// Mitsubishi GX Works2 project: Ex5   PLC: Q03UDV

PROGRAM MAIN
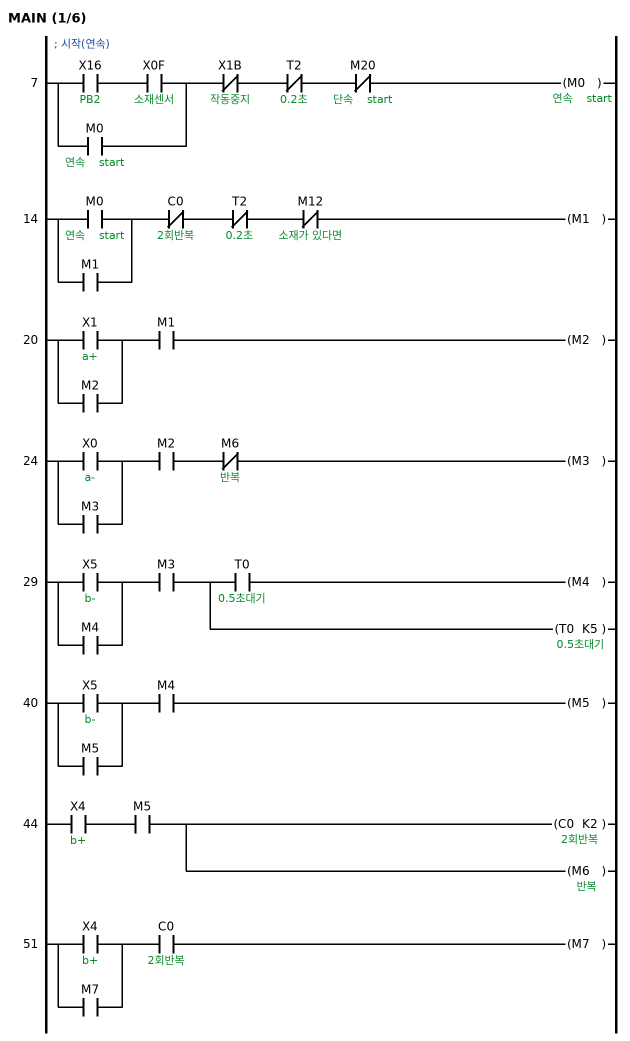
; 시작(연속)
7     LD      X16  ; PB2
      AND     X0F  ; 소재센서
      OR      M0  ; 연속    start
      ANI     X1B  ; 작동중지
      ANI     T2  ; 0.2초
      ANI     M20  ; 단속    start
      OUT     M0  ; 연속    start
14    LD      M0  ; 연속    start
      OR      M1
      ANI     C0  ; 2회반복
      ANI     T2  ; 0.2초
      ANI     M12  ; 소재가 있다면
      OUT     M1
20    LD      X1  ; a+
      OR      M2
      AND     M1
      OUT     M2
24    LD      X0  ; a-
      OR      M3
      AND     M2
      ANI     M6  ; 반복
      OUT     M3
29    LD      X5  ; b-
      OR      M4
      AND     M3
      MPS
      AND     T0  ; 0.5초대기
      OUT     M4
      MPP
      OUT     T0 K5  ; 0.5초대기
40    LD      X5  ; b-
      OR      M5
      AND     M4
      OUT     M5
44    LD      X4  ; b+
      AND     M5
      OUT     C0 K2  ; 2회반복
      OUT     M6  ; 반복
51    LD      X4  ; b+
      OR      M7
      AND     C0  ; 2회반복
      OUT     M7
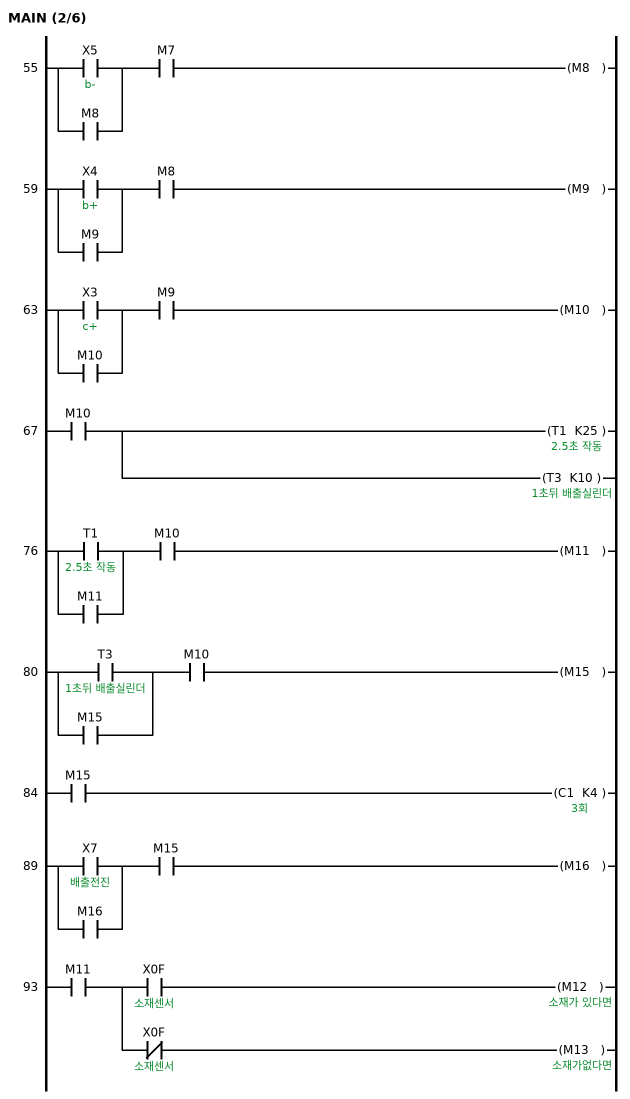
55    LD      X5  ; b-
      OR      M8
      AND     M7
      OUT     M8
59    LD      X4  ; b+
      OR      M9
      AND     M8
      OUT     M9
63    LD      X3  ; c+
      OR      M10
      AND     M9
      OUT     M10
67    LD      M10
      OUT     T1 K25  ; 2.5초 작동
      OUT     T3 K10  ; 1초뒤 배출실린더
76    LD      T1  ; 2.5초 작동
      OR      M11
      AND     M10
      OUT     M11
80    LD      T3  ; 1초뒤 배출실린더
      OR      M15
      AND     M10
      OUT     M15
84    LD      M15
      OUT     C1 K4  ; 3회
89    LD      X7  ; 배출전진
      OR      M16
      AND     M15
      OUT     M16
93    LD      M11
      MPS
      AND     X0F  ; 소재센서
      OUT     M12  ; 소재가 있다면
      MPP
      ANI     X0F  ; 소재센서
      OUT     M13  ; 소재가없다면
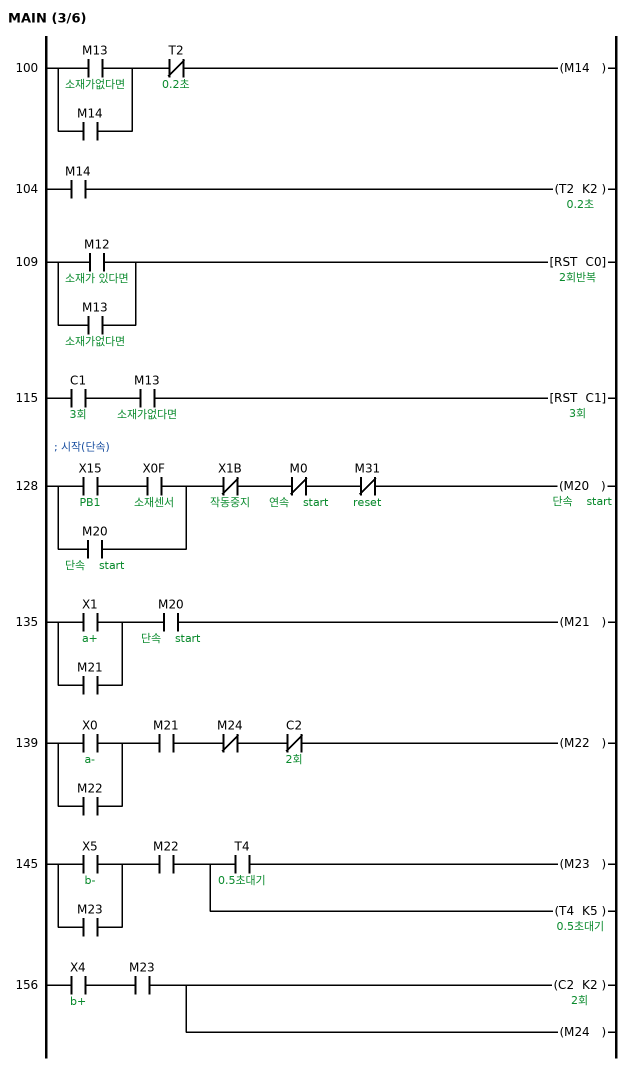
100   LD      M13  ; 소재가없다면
      OR      M14
      ANI     T2  ; 0.2초
      OUT     M14
104   LD      M14
      OUT     T2 K2  ; 0.2초
109   LD      M12  ; 소재가 있다면
      OR      M13  ; 소재가없다면
      RST     C0  ; 2회반복
115   LD      C1  ; 3회
      AND     M13  ; 소재가없다면
      RST     C1  ; 3회
; 시작(단속)
128   LD      X15  ; PB1
      AND     X0F  ; 소재센서
      OR      M20  ; 단속    start
      ANI     X1B  ; 작동중지
      ANI     M0  ; 연속    start
      ANI     M31  ; reset
      OUT     M20  ; 단속    start
135   LD      X1  ; a+
      OR      M21
      AND     M20  ; 단속    start
      OUT     M21
139   LD      X0  ; a-
      OR      M22
      AND     M21
      ANI     M24
      ANI     C2  ; 2회
      OUT     M22
145   LD      X5  ; b-
      OR      M23
      AND     M22
      MPS
      AND     T4  ; 0.5초대기
      OUT     M23
      MPP
      OUT     T4 K5  ; 0.5초대기
156   LD      X4  ; b+
      AND     M23
      OUT     C2 K2  ; 2회
      OUT     M24
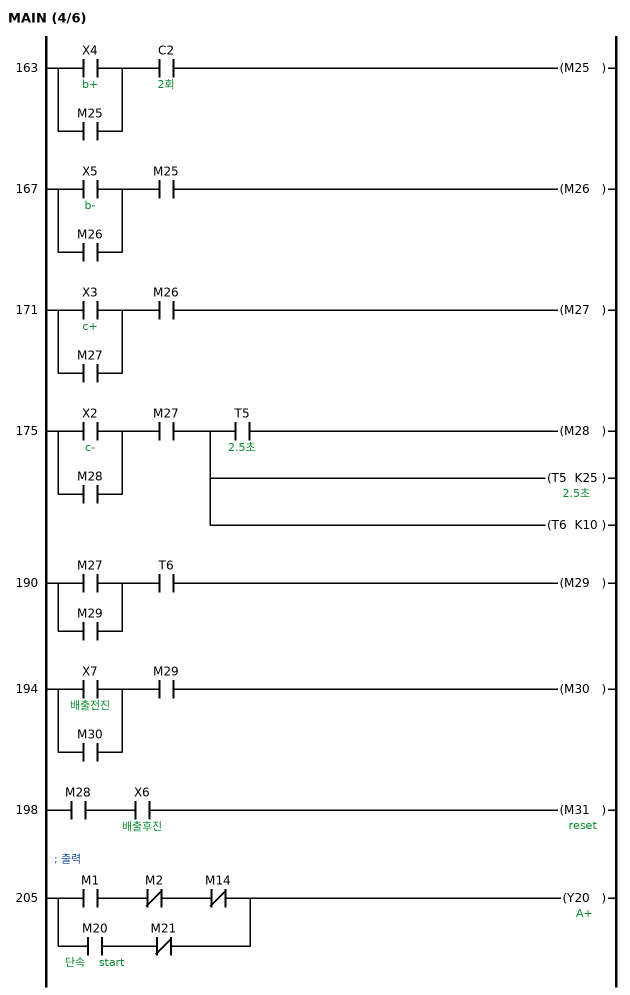
163   LD      X4  ; b+
      OR      M25
      AND     C2  ; 2회
      OUT     M25
167   LD      X5  ; b-
      OR      M26
      AND     M25
      OUT     M26
171   LD      X3  ; c+
      OR      M27
      AND     M26
      OUT     M27
175   LD      X2  ; c-
      OR      M28
      AND     M27
      MPS
      AND     T5  ; 2.5초
      OUT     M28
      MPP
      OUT     T5 K25  ; 2.5초
      OUT     T6 K10
190   LD      M27
      OR      M29
      AND     T6
      OUT     M29
194   LD      X7  ; 배출전진
      OR      M30
      AND     M29
      OUT     M30
198   LD      M28
      AND     X6  ; 배출후진
      OUT     M31  ; reset
; 출력
205   LD      M1
      ANI     M2
      ANI     M14
      LD      M20  ; 단속    start
      ANI     M21
      ORB
      OUT     Y20  ; A+
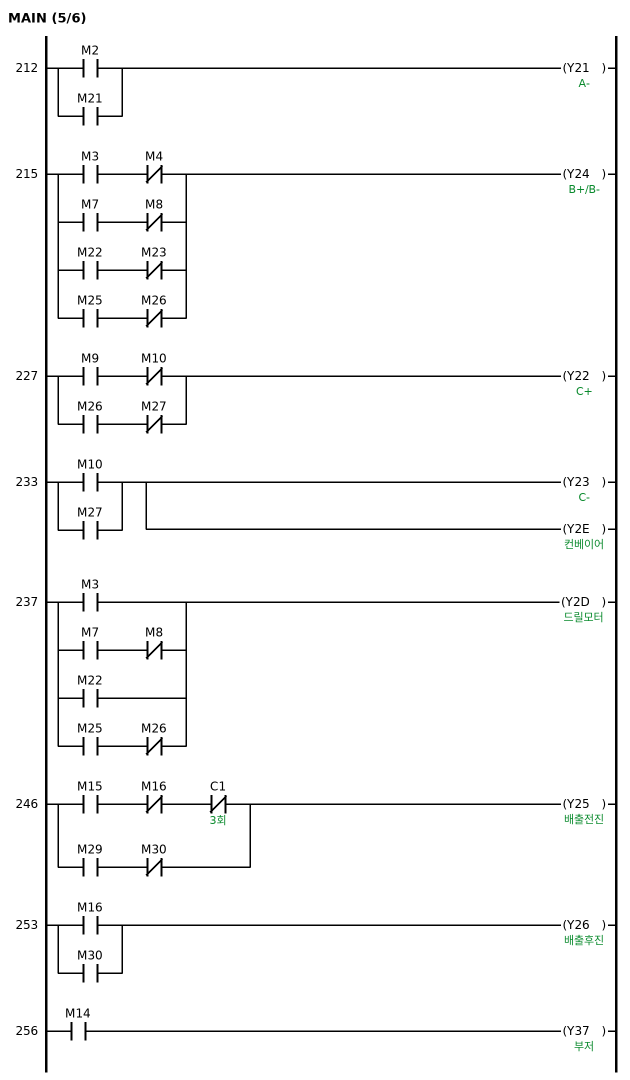
212   LD      M2
      OR      M21
      OUT     Y21  ; A-
215   LD      M3
      ANI     M4
      LD      M7
      ANI     M8
      ORB
      LD      M22
      ANI     M23
      ORB
      LD      M25
      ANI     M26
      ORB
      OUT     Y24  ; B+/B-
227   LD      M9
      ANI     M10
      LD      M26
      ANI     M27
      ORB
      OUT     Y22  ; C+
233   LD      M10
      OR      M27
      OUT     Y23  ; C-
      OUT     Y2E  ; 컨베이어
237   LD      M3
      LD      M7
      ANI     M8
      ORB
      OR      M22
      LD      M25
      ANI     M26
      ORB
      OUT     Y2D  ; 드릴모터
246   LD      M15
      ANI     M16
      ANI     C1  ; 3회
      LD      M29
      ANI     M30
      ORB
      OUT     Y25  ; 배출전진
253   LD      M16
      OR      M30
      OUT     Y26  ; 배출후진
256   LD      M14
      OUT     Y37  ; 부저
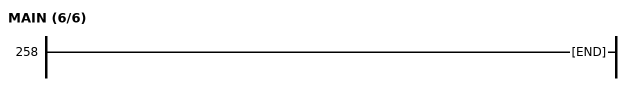
258   END
END_PROGRAM
